// TIA Portal V19 export
VAR_GLOBAL   // PLC tag table "EM120_Template"
END_VAR
VAR_GLOBAL CONSTANT   // user constants
   NMAX_ERROR_NOREACTION_EM120 : Int := 1;   // Number of Error (no reaction) type alarms
   NMAX_ERROR_ABORT_EM120 : Int := 1;   // Number of Error (command abort) type alarms
   NMAX_ERROR_STOP_EM120 : Int := 50;   // Number of Error (command stop) type alarms
   NMAX_WARNING_NOREACTION_EM120 : Int := 1;   // Number of Warning (no reaction) type alarms
   NMAX_WARNING_HOLD_EM120 : Int := 1;   // Number of Warning (command hold) type alarms
   NMAX_WARNING_SUSPEND_EM120 : Int := 1;   // Number of Warning (command suspend) type alarms
   NMAX_INFORMATION_EM120 : Int := 1;   // Number of Information type alarms
   NMAX_CRITERIAANALYSIS_EM120 : Int := 1;   // Criteria analysis
END_VAR
